FUNCTION_BLOCK FB_MotionStageNCParams
(*
    Read and refresh axis parameters struct on ST_MotionStage
*)
VAR_IN_OUT
    stMotionStage: ST_MotionStage;
END_VAR
VAR_INPUT
    bEnable: BOOL;
    tRefreshDelay: TIME;
END_VAR
VAR_OUTPUT
    bError: BOOL;
END_VAR
VAR
    mcReadParams: MC_ReadParameterSet;
    timer: TON;
    bExecute: BOOL := TRUE;
    nLatchErrId: UDINT;
END_VAR

timer(
    IN:=bEnable AND NOT bExecute,
    PT:=tRefreshDelay);
bExecute S= timer.Q;
mcReadParams(
    Parameter:=stMotionStage.stAxisParameters,
    Axis:=stMotionStage.Axis,
    Execute:=bEnable AND bExecute,
    Error=>bError);
IF mcReadParams.ErrorID <> 0 THEN
    nLatchErrId := 0;
END_IF
bExecute R= mcReadParams.Done OR mcReadParams.Error;
stMotionStage.bAxisParamsInit S= mcReadParams.Done;

END_FUNCTION_BLOCK

(* stored: Version 1.1.0.1, ProductVersion 3.1.4022.18
   POU FB_MotionStageNCParams: Id {ffafdde1-c9c9-04ad-2047-9434c7439ed8}, SpecialFunc None *)
